(* PLC project Unnamed, Unknown Unnamed 1 *)
(* stored: creationDateTime 2023-03-30T14:33:54, modificationDateTime 2023-04-18T10:15:01 *)

PROGRAM slave_device
  VAR
    Send_Slave AT %IX0.0 : BOOL := 0;
    Recieve_Slave AT %IX100.0 : BOOL := 0;
    Switch AT %QX0.0 : BOOL;
    LED AT %QX100.0 : BOOL;
  END_VAR
  VAR
    TON0 : TON;
    TOF0 : TOF;
    TON1 : TON;
    TOF1 : TOF;
  END_VAR

(* LD diagram, written out as Structured Text *)
TON0(IN := NOT Switch AND NOT Send_Slave, PT := T#1000ms);
TOF0(EN := TON0.ENO, IN := TON0.Q, PT := T#1000ms);
Switch := TOF0.Q;
TON1(IN := NOT LED AND NOT Recieve_Slave, PT := T#1000ms);
TOF1(EN := TON1.ENO, IN := TON1.Q, PT := T#1000ms);
LED := TOF1.Q;
END_PROGRAM

CONFIGURATION Config0
  RESOURCE Res0 ON PLC
    TASK task0(INTERVAL := T#100ms, PRIORITY := 0);
    PROGRAM instance0 WITH task0 : slave_device;
  END_RESOURCE
END_CONFIGURATION
